// Mitsubishi GX Works2 project: BookEX6_23 Arithmetic   PLC: Q13UDV

// global labels: Global
VAR_GLOBAL
  bVar0 AT M5000 : BOOL;
  abArray0 AT M5010 : ARRAY [0..49] OF BOOL;
  sStr0 AT D5000 : STRING[199];
  sStr1 AT D5100 : STRING[199];
  sStr2 AT D5200 : STRING[199];
  sStr3 AT D5300 : STRING[199];
  sStr4 AT D5400 : STRING[199];
  sStr5 AT D5500 : STRING[199];
  sStr6 AT D5600 : STRING[199];
  sStr7 AT D5700 : STRING[199];
  sStr8 AT D5800 : STRING[199];
  sStr9 AT D5900 : STRING[199];
  iVar0 AT D4500 : INT;
  iVar1 AT D4501 : INT;
  iVar2 AT D4502 : INT;
  iVar3 AT D4503 : INT;
  iVar4 AT D4504 : INT;
  iVar5 AT D4505 : INT;
  iVar6 AT D4506 : INT;
  iVar7 AT D4507 : INT;
  iVar8 AT D4508 : INT;
  iVar9 AT D4509 : INT;
  dVar0 AT D4510 : DINT;
  dVar1 AT D4512 : DINT;
  dVar2 AT D4514 : DINT;
  dVar3 AT D4516 : DINT;
  dVar4 AT D4518 : DINT;
  dVar5 AT D4520 : DINT;
  dVar6 AT D4522 : DINT;
  dVar7 AT D4524 : DINT;
  dVar8 AT D4526 : DINT;
  dVar9 AT D4528 : DINT;
  wVar0 AT D4530 : WORD;
  wVar1 AT D4531 : WORD;
  wVar2 AT D4532 : WORD;
  wVar3 AT D4533 : WORD;
  wVar4 AT D4534 : WORD;
  wVar5 AT D4535 : WORD;
  wVar6 AT D4536 : WORD;
  wVar7 AT D4537 : WORD;
  wVar8 AT D4538 : WORD;
  wVar9 AT D4539 : WORD;
  dwVar0 AT D4540 : DWORD;
  dwVar1 AT D4542 : DWORD;
  dwVar2 AT D4544 : DWORD;
  dwVar3 AT D4546 : DWORD;
  dwVar4 AT D4548 : DWORD;
  dwVar5 AT D4550 : DWORD;
  dwVar6 AT D4552 : DWORD;
  dwVar7 AT D4554 : DWORD;
  dwVar8 AT D4556 : DWORD;
  dwVar9 AT D4558 : DWORD;
  fsVar0 AT D4560 : REAL;
  fsVar1 AT D4562 : REAL;
  fsVar2 AT D4564 : REAL;
  fsVar3 AT D4566 : REAL;
  fsVar4 AT D4568 : REAL;
  fsVar5 AT D4570 : REAL;
  fsVar6 AT D4572 : REAL;
  fsVar7 AT D4574 : REAL;
  fsVar8 AT D4576 : REAL;
  fsVar9 AT D4578 : REAL;
  fdVar0 AT D4580 : LREAL;
  tTime0 AT D4620 : TIME;
  tTime1 AT D4622 : TIME;
  tTime2 AT D4624 : TIME;
  tTime3 AT D4626 : TIME;
  tTime4 AT D4628 : TIME;
  tTime5 AT D4630 : TIME;
  tTime6 AT D4632 : TIME;
  tTime7 AT D4634 : TIME;
  tTime8 AT D4636 : TIME;
  tTime9 AT D4638 : TIME;
  tTime10 AT D4640 : TIME;
  bVar1 AT M5001 : BOOL;
  bVar2 AT M5002 : BOOL;
  bVar3 AT M5003 : BOOL;
  bVar4 AT M5004 : BOOL;
  bVar5 AT M5005 : BOOL;
  bVar6 AT M5006 : BOOL;
  bVar7 AT M5007 : BOOL;
  bVar8 AT M5008 : BOOL;
  bVar9 AT M5009 : BOOL;
  abArray1 AT M5060 : ARRAY [0..49] OF BOOL;
  abArray2 AT M5110 : ARRAY [0..49] OF BOOL;
  abArray3 AT M5160 : ARRAY [0..49] OF BOOL;
  abArray4 AT M5210 : ARRAY [0..49] OF BOOL;
  abArray5 AT M5260 : ARRAY [0..49] OF BOOL;
  abArray6 AT M5310 : ARRAY [0..49] OF BOOL;
  abArray7 AT M5360 : ARRAY [0..49] OF BOOL;
  abArray8 AT M5410 : ARRAY [0..49] OF BOOL;
  abArray9 AT M5460 : ARRAY [0..49] OF BOOL;
  fdVar1 AT D4584 : LREAL;
  fdVar2 AT D4588 : LREAL;
  fdVar3 AT D4592 : LREAL;
  fdVar4 AT D4596 : LREAL;
  fdVar5 AT D4600 : LREAL;
  fdVar6 AT D4604 : LREAL;
  fdVar7 AT D4608 : LREAL;
  fdVar8 AT D4612 : LREAL;
  fdVar9 AT D4616 : LREAL;
  afsPen0 AT D2000 : ARRAY [0..499] OF REAL;
  afsPen1 AT D3000 : ARRAY [0..499] OF REAL;
END_VAR
// user libraries (not included): HMI

PROGRAM ExAddSub2
VAR
  HMI20_1 : HMI20;
END_VAR
(* structured ladder/FBD written out as ST: instructions are called as NAME(EN, inputs, outputs); _pN, _eN, _tN stand for wires *)
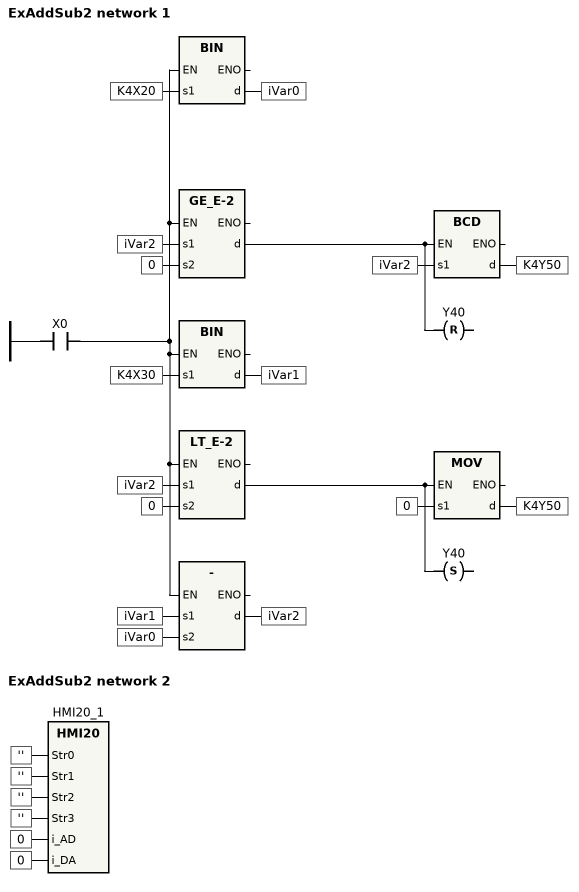
(* network 1 *)
BIN(X0, K4X20, iVar0);
BIN(X0, K4X30, iVar1);
-(X0, iVar1, iVar0, iVar2);
GE_E(X0, iVar2, 0, _t1);
BCD(_t1, iVar2, K4Y50);
RST(_t1, Y40);
LT_E(X0, iVar2, 0, _t2);
SET(_t2, Y40);
MOV(_t2, 0, K4Y50);
(* network 2 *)
HMI20_1(Str0 := '', Str1 := '', Str2 := '', Str3 := '', i_AD := 0, i_DA := 0);
END_PROGRAM

PROGRAM ExB
VAR
  wVar20 : WORD;
  wVar21 : WORD;
  wVar22 : WORD;
  wVar23 : WORD;
  wVar24 : WORD;
  wVar25 : WORD;
  wVar26 : WORD;
  wVar27 : WORD;
  wVar28 : WORD;
  wVar29 : WORD;
  dwVar20 : DWORD;
  dwVar21 : DWORD;
  dwVar22 : DWORD;
  dwVar23 : DWORD;
  dwVar24 : DWORD;
  dwVar25 : DWORD;
  dwVar26 : DWORD;
  dwVar27 : DWORD;
  dwVar28 : DWORD;
  dwVar29 : DWORD;
  awVar0 : ARRAY [0..1] OF WORD;
  awVar1 : ARRAY [0..1] OF WORD;
  awVar2 : ARRAY [0..3] OF WORD;
  awVar3 : ARRAY [0..3] OF WORD;
  adwVar3 : ARRAY [0..1] OF DWORD;
END_VAR
(* structured ladder/FBD written out as ST: instructions are called as NAME(EN, inputs, outputs); _pN, _eN, _tN stand for wires *)
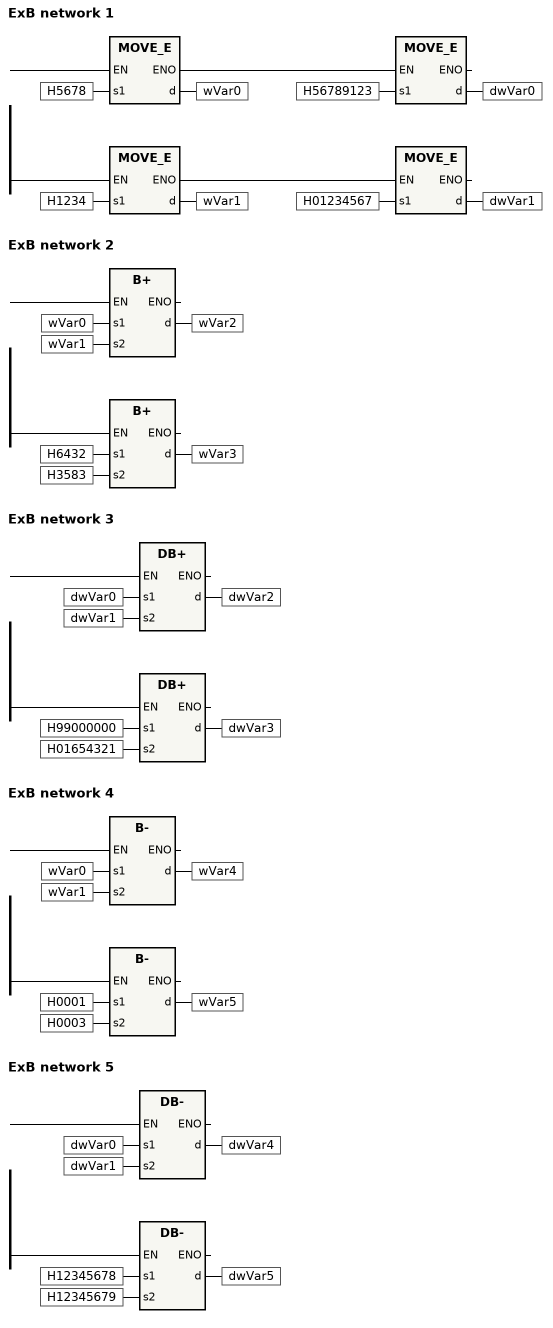
(* network 1 *)
_e1 := MOVE_E(TRUE, H5678, wVar0);
MOVE_E(_e1, H56789123, dwVar0);
_e2 := MOVE_E(TRUE, H1234, wVar1);
MOVE_E(_e2, H01234567, dwVar1);
(* network 2 *)
B+(TRUE, wVar0, wVar1, wVar2);
B+(TRUE, H6432, H3583, wVar3);
(* network 3 *)
DB+(TRUE, dwVar0, dwVar1, dwVar2);
DB+(TRUE, H99000000, H01654321, dwVar3);
(* network 4 *)
B-(TRUE, wVar0, wVar1, wVar4);
B-(TRUE, H0001, H0003, wVar5);
(* network 5 *)
DB-(TRUE, dwVar0, dwVar1, dwVar4);
DB-(TRUE, H12345678, H12345679, dwVar5);
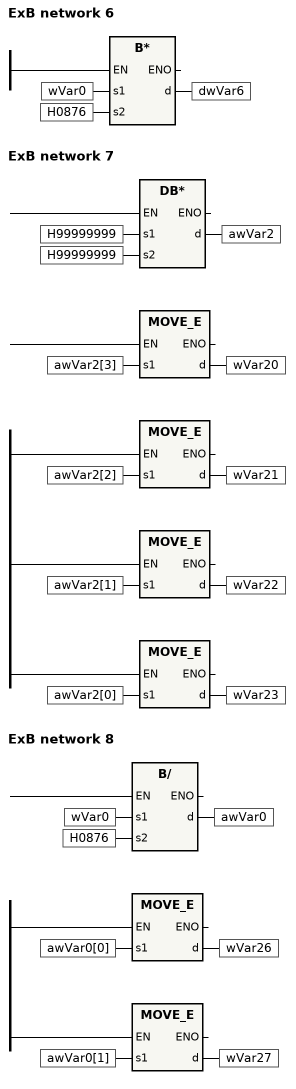
(* network 6 *)
B*(TRUE, wVar0, H0876, dwVar6);
(* network 7 *)
DB*(TRUE, H99999999, H99999999, awVar2);
MOVE_E(TRUE, awVar2[3], wVar20);
MOVE_E(TRUE, awVar2[2], wVar21);
MOVE_E(TRUE, awVar2[1], wVar22);
MOVE_E(TRUE, awVar2[0], wVar23);
(* network 8 *)
B/(TRUE, wVar0, H0876, awVar0);
MOVE_E(TRUE, awVar0[0], wVar26);
MOVE_E(TRUE, awVar0[1], wVar27);
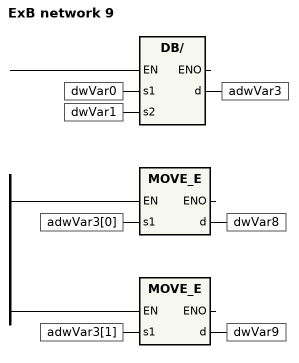
(* network 9 *)
DB/(TRUE, dwVar0, dwVar1, adwVar3);
MOVE_E(TRUE, adwVar3[0], dwVar8);
MOVE_E(TRUE, adwVar3[1], dwVar9);
END_PROGRAM

PROGRAM ExBK
VAR
  Mov4INT_1 : Mov4INT;
  Mov4INT_2 : Mov4INT;
END_VAR
(* structured ladder/FBD written out as ST: instructions are called as NAME(EN, inputs, outputs); _pN, _eN, _tN stand for wires *)
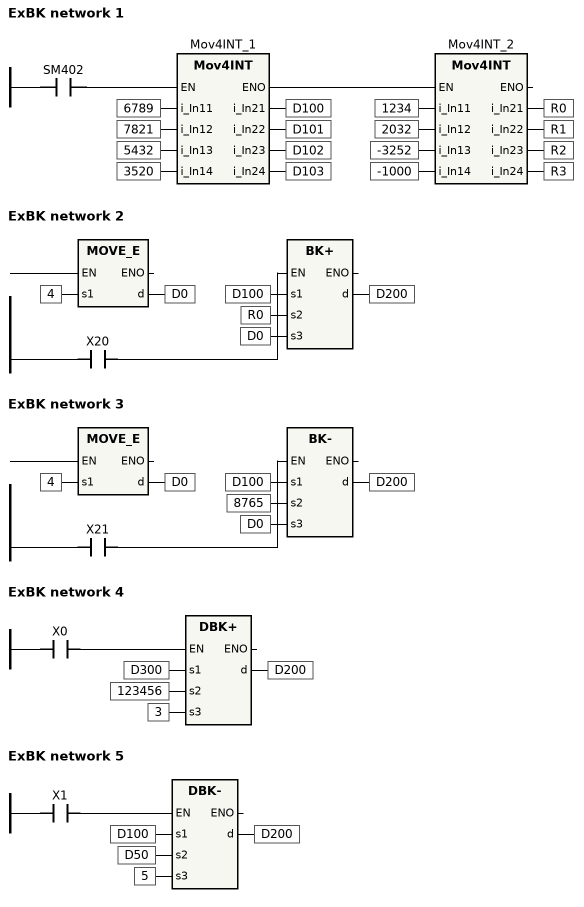
(* network 1 *)
Mov4INT_1(EN := SM402, i_In11 := 6789, i_In12 := 7821, i_In13 := 5432, i_In14 := 3520, i_In21 => D100, i_In22 => D101, i_In23 => D102, i_In24 => D103);
Mov4INT_2(EN := Mov4INT_1.ENO, i_In11 := 1234, i_In12 := 2032, i_In13 := -3252, i_In14 := -1000, i_In21 => R0, i_In22 => R1, i_In23 => R2, i_In24 => R3);
(* network 2 *)
MOVE_E(TRUE, 4, D0);
BK+(X20, D100, R0, D0, D200);
(* network 3 *)
MOVE_E(TRUE, 4, D0);
BK-(X21, D100, 8765, D0, D200);
(* network 4 *)
DBK+(X0, D300, 123456, 3, D200);
(* network 5 *)
DBK-(X1, D100, D50, 5, D200);
END_PROGRAM

PROGRAM ExIncDec
(* structured ladder/FBD written out as ST: instructions are called as NAME(EN, inputs, outputs); _pN, _eN, _tN stand for wires *)
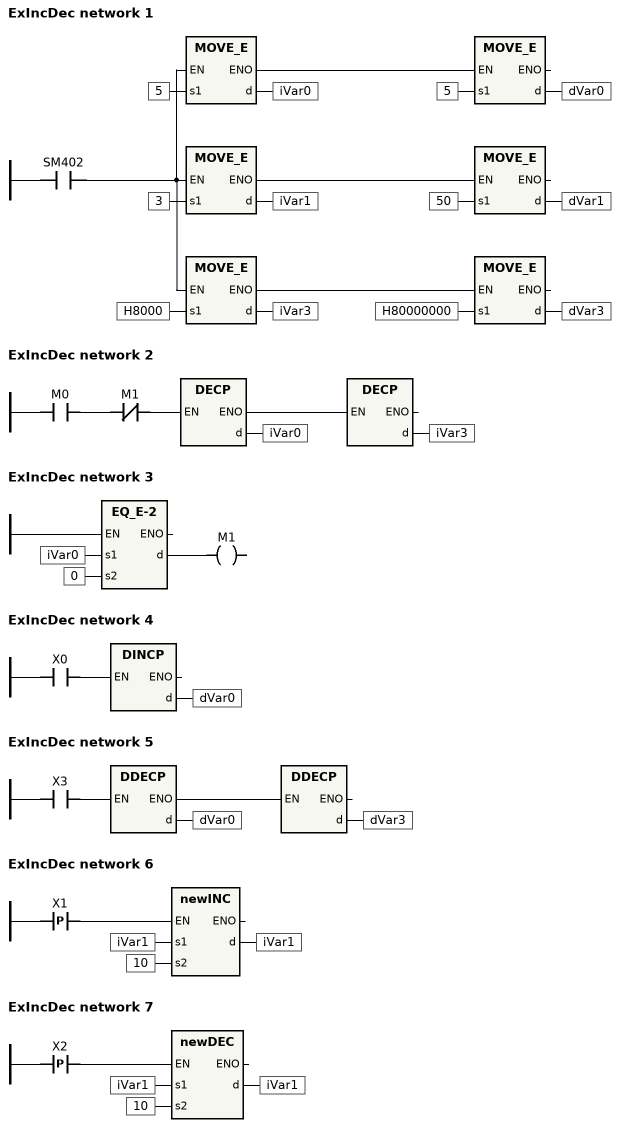
(* network 1 *)
_e1 := MOVE_E(SM402, 5, iVar0);
MOVE_E(_e1, 5, dVar0);
_e2 := MOVE_E(SM402, 3, iVar1);
MOVE_E(_e2, 50, dVar1);
_e3 := MOVE_E(SM402, H8000, iVar3);
MOVE_E(_e3, H80000000, dVar3);
(* network 2 *)
_e1 := DECP(M0 AND NOT M1, iVar0);
DECP(_e1, iVar3);
(* network 3 *)
EQ_E(TRUE, iVar0, 0, _t1);
M1 := _t1;
(* network 4 *)
DINCP(X0, dVar0);
(* network 5 *)
_e1 := DDECP(X3, dVar0);
DDECP(_e1, dVar3);
(* network 6 *)
newINC(LDP(TRUE, X1), iVar1, 10, iVar1);
(* network 7 *)
newDEC(LDP(TRUE, X2), iVar1, 10, iVar1);
END_PROGRAM

PROGRAM ExMulDiv
VAR
  iVar20 : INT;
  iVar21 : INT;
  iVar22 : INT;
  iVar23 : INT;
  iVar24 : INT;
  iVar25 : INT;
  iVar26 : INT;
  iVar27 : INT;
  iVar28 : INT;
  iVar29 : INT;
  dVar20 : DINT;
  dVar21 : DINT;
  dVar22 : DINT;
  dVar23 : DINT;
  dVar24 : DINT;
  dVar25 : DINT;
  dVar26 : DINT;
  dVar27 : DINT;
  dVar28 : DINT;
  dVar29 : DINT;
  aiVar0 : ARRAY [0..1] OF INT;
  aiVar1 : ARRAY [0..1] OF INT;
  aiVar2 : ARRAY [0..2] OF INT;
  awVar0 : ARRAY [0..1] OF WORD;
  awVar1 : ARRAY [0..1] OF WORD;
  awVar2 : ARRAY [0..3] OF WORD;
  awVar3 : ARRAY [0..3] OF WORD;
  adwVar3 : ARRAY [0..1] OF DWORD;
  adVar0 : ARRAY [0..1] OF DINT;
  adVar1 : ARRAY [0..1] OF DINT;
  adVar2 : ARRAY [0..1] OF DINT;
  adVar3 : ARRAY [0..1] OF DINT;
  adVar4 : ARRAY [0..1] OF DINT;
END_VAR
(* structured ladder/FBD written out as ST: instructions are called as NAME(EN, inputs, outputs); _pN, _eN, _tN stand for wires *)
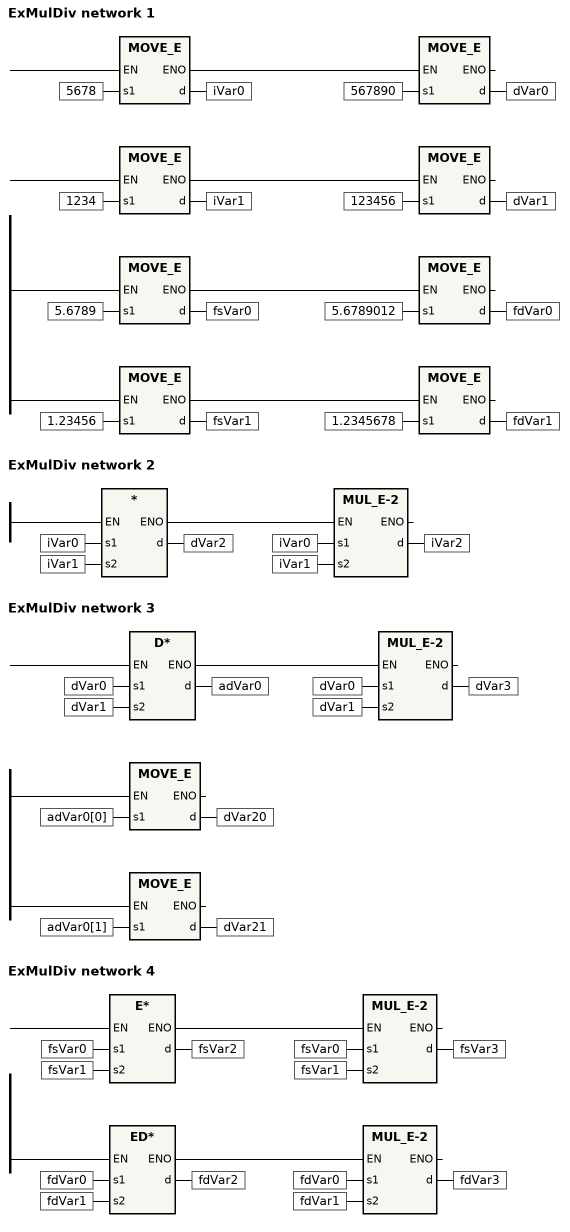
(* network 1 *)
_e1 := MOVE_E(TRUE, 5678, iVar0);
MOVE_E(_e1, 567890, dVar0);
_e2 := MOVE_E(TRUE, 1234, iVar1);
MOVE_E(_e2, 123456, dVar1);
_e3 := MOVE_E(TRUE, 5.6789, fsVar0);
MOVE_E(_e3, 5.6789012, fdVar0);
_e4 := MOVE_E(TRUE, 1.23456, fsVar1);
MOVE_E(_e4, 1.2345678, fdVar1);
(* network 2 *)
_e1 := *(TRUE, iVar0, iVar1, dVar2);
MUL_E(_e1, iVar0, iVar1, iVar2);
(* network 3 *)
_e1 := D*(TRUE, dVar0, dVar1, adVar0);
MUL_E(_e1, dVar0, dVar1, dVar3);
MOVE_E(TRUE, adVar0[0], dVar20);
MOVE_E(TRUE, adVar0[1], dVar21);
(* network 4 *)
_e1 := E*(TRUE, fsVar0, fsVar1, fsVar2);
MUL_E(_e1, fsVar0, fsVar1, fsVar3);
_e2 := ED*(TRUE, fdVar0, fdVar1, fdVar2);
MUL_E(_e2, fdVar0, fdVar1, fdVar3);
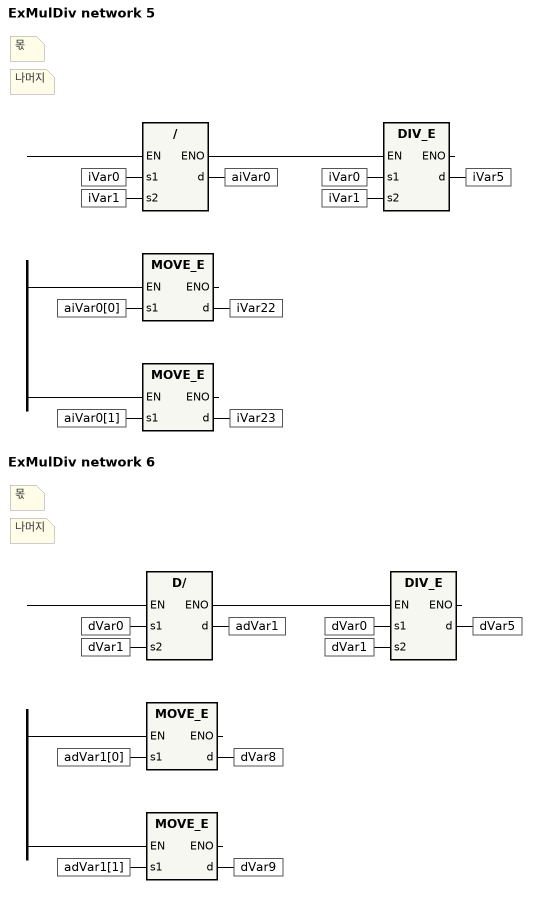
(* network 5 *)
(* 몫 *)
(* 나머지 *)
_e1 := /(TRUE, iVar0, iVar1, aiVar0);
DIV_E(_e1, iVar0, iVar1, iVar5);
MOVE_E(TRUE, aiVar0[0], iVar22);
MOVE_E(TRUE, aiVar0[1], iVar23);
(* network 6 *)
(* 몫 *)
(* 나머지 *)
_e1 := D/(TRUE, dVar0, dVar1, adVar1);
DIV_E(_e1, dVar0, dVar1, dVar5);
MOVE_E(TRUE, adVar1[0], dVar8);
MOVE_E(TRUE, adVar1[1], dVar9);
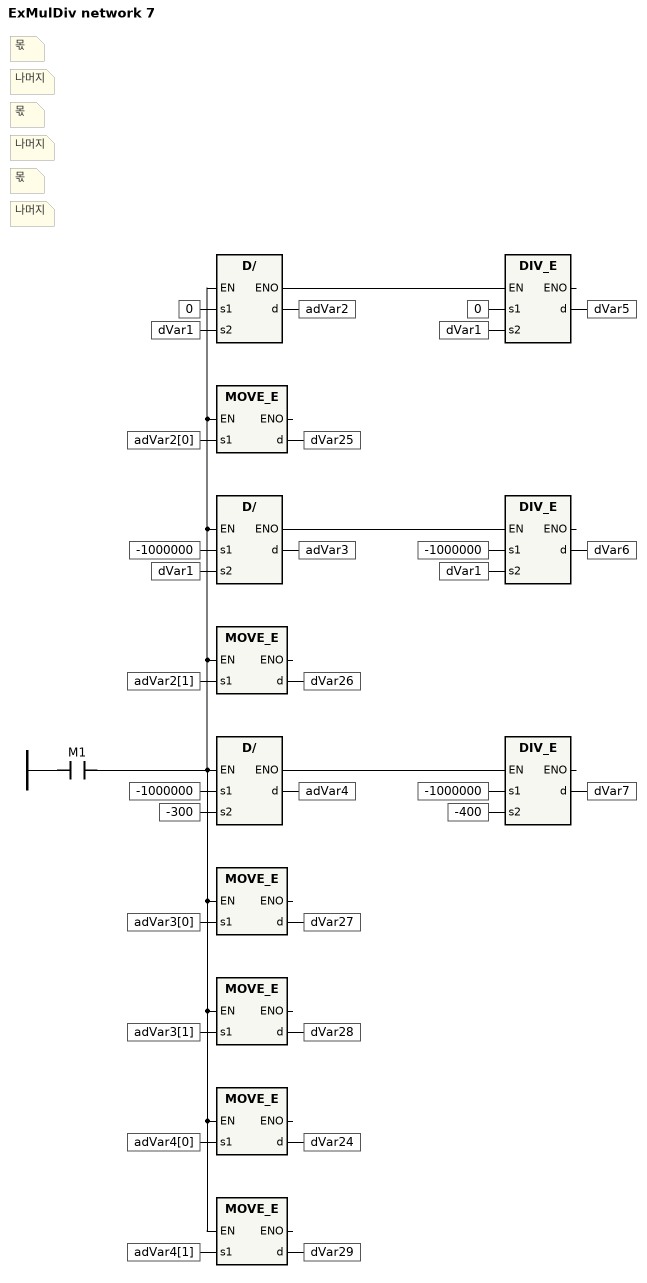
(* network 7 *)
(* 몫 *)
(* 나머지 *)
(* 몫 *)
(* 나머지 *)
(* 몫 *)
(* 나머지 *)
_e1 := D/(M1, 0, dVar1, adVar2);
DIV_E(_e1, 0, dVar1, dVar5);
MOVE_E(M1, adVar2[0], dVar25);
MOVE_E(M1, adVar2[1], dVar26);
_e2 := D/(M1, -1000000, dVar1, adVar3);
DIV_E(_e2, -1000000, dVar1, dVar6);
MOVE_E(M1, adVar3[0], dVar27);
MOVE_E(M1, adVar3[1], dVar28);
_e3 := D/(M1, -1000000, -300, adVar4);
DIV_E(_e3, -1000000, -400, dVar7);
MOVE_E(M1, adVar4[0], dVar24);
MOVE_E(M1, adVar4[1], dVar29);
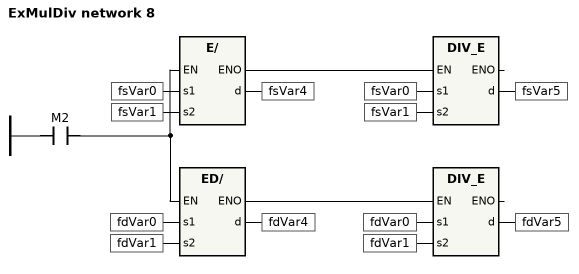
(* network 8 *)
_e1 := E/(M2, fsVar0, fsVar1, fsVar4);
DIV_E(_e1, fsVar0, fsVar1, fsVar5);
_e2 := ED/(M2, fdVar0, fdVar1, fdVar4);
DIV_E(_e2, fdVar0, fdVar1, fdVar5);
END_PROGRAM

PROGRAM ExString
(* structured ladder/FBD written out as ST: instructions are called as NAME(EN, inputs, outputs); _pN, _eN, _tN stand for wires *)
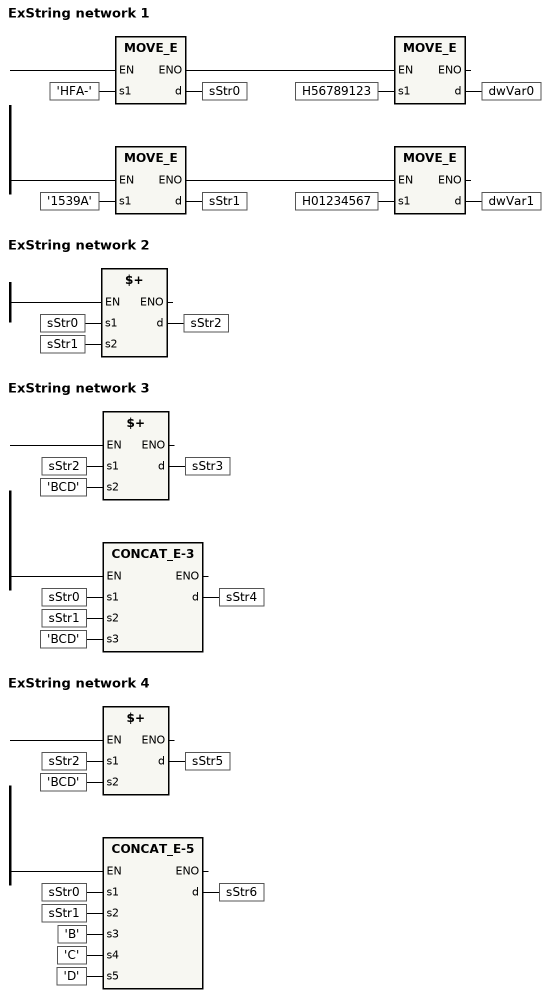
(* network 1 *)
_e1 := MOVE_E(TRUE, 'HFA-', sStr0);
MOVE_E(_e1, H56789123, dwVar0);
_e2 := MOVE_E(TRUE, '1539A', sStr1);
MOVE_E(_e2, H01234567, dwVar1);
(* network 2 *)
$+(TRUE, sStr0, sStr1, sStr2);
(* network 3 *)
$+(TRUE, sStr2, 'BCD', sStr3);
CONCAT_E(TRUE, sStr0, sStr1, 'BCD', sStr4);
(* network 4 *)
$+(TRUE, sStr2, 'BCD', sStr5);
CONCAT_E(TRUE, sStr0, sStr1, 'B', 'C', 'D', sStr6);
END_PROGRAM

FUNCTION newDEC
VAR_INPUT
  i_IN : INT;
  i_Max : INT;
END_VAR
VAR
  ix : INT;
END_VAR
;
ix := i_IN - 1;
IF ix < 0 THEN
	ix := i_Max;
END_IF;
newDEC := ix;
END_FUNCTION

FUNCTION newINC
VAR_INPUT
  i_IN : INT;
  i_Max : INT;
END_VAR
VAR
  ix : INT;
END_VAR
;
ix := i_IN + 1;
IF ix > i_Max THEN
	ix := 0;
END_IF;
newINC := ix;
END_FUNCTION

PROGRAM ExIncDec2
(* structured ladder/FBD written out as ST: instructions are called as NAME(EN, inputs, outputs); _pN, _eN, _tN stand for wires *)
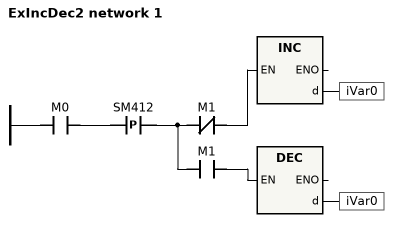
(* network 1 *)
_p1 := M0 AND LDP(TRUE, SM412);
INC(_p1 AND NOT M1, iVar0);
DEC(_p1 AND M1, iVar0);
END_PROGRAM

PROGRAM ExAddSub
VAR
  iVar20 : INT;
  iVar21 : INT;
  iVar22 : INT;
  iVar23 : INT;
  iVar24 : INT;
  iVar25 : INT;
  iVar26 : INT;
  iVar27 : INT;
  iVar28 : INT;
  iVar29 : INT;
  dVar20 : DINT;
  dVar21 : DINT;
  dVar22 : DINT;
  dVar23 : DINT;
  dVar24 : DINT;
  dVar25 : DINT;
  dVar26 : DINT;
  dVar27 : DINT;
  dVar28 : DINT;
  dVar29 : DINT;
  HMI05_1 : HMI05;
END_VAR
(* structured ladder/FBD written out as ST: instructions are called as NAME(EN, inputs, outputs); _pN, _eN, _tN stand for wires *)
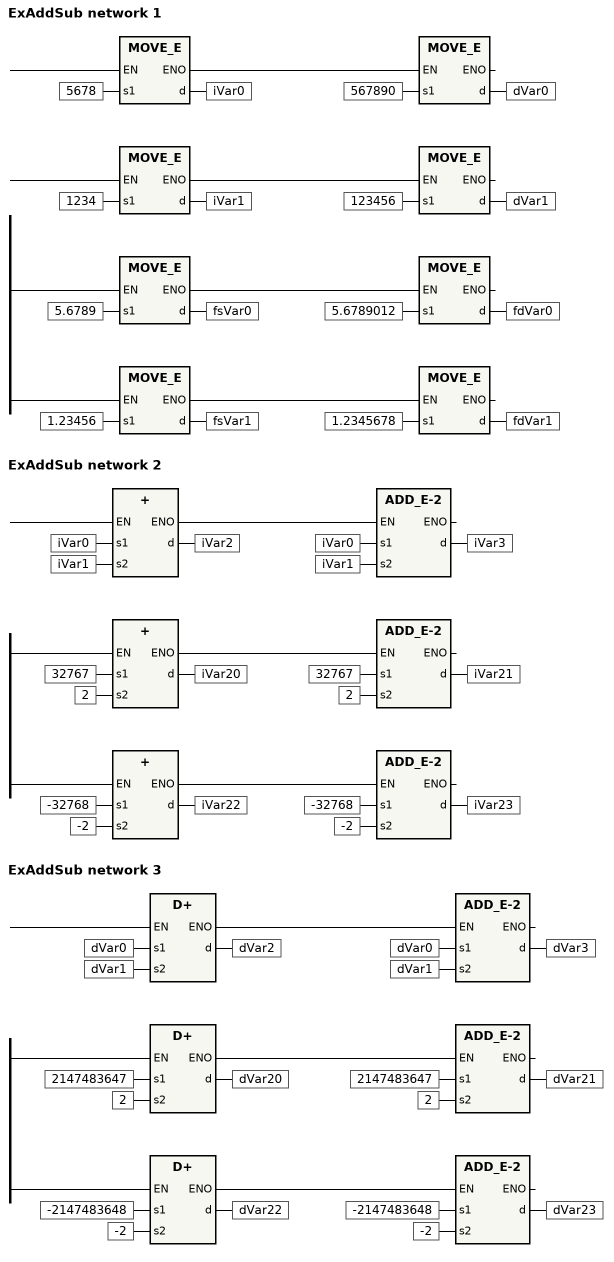
(* network 1 *)
_e1 := MOVE_E(TRUE, 5678, iVar0);
MOVE_E(_e1, 567890, dVar0);
_e2 := MOVE_E(TRUE, 1234, iVar1);
MOVE_E(_e2, 123456, dVar1);
_e3 := MOVE_E(TRUE, 5.6789, fsVar0);
MOVE_E(_e3, 5.6789012, fdVar0);
_e4 := MOVE_E(TRUE, 1.23456, fsVar1);
MOVE_E(_e4, 1.2345678, fdVar1);
(* network 2 *)
_e1 := +(TRUE, iVar0, iVar1, iVar2);
ADD_E(_e1, iVar0, iVar1, iVar3);
_e2 := +(TRUE, 32767, 2, iVar20);
ADD_E(_e2, 32767, 2, iVar21);
_e3 := +(TRUE, -32768, -2, iVar22);
ADD_E(_e3, -32768, -2, iVar23);
(* network 3 *)
_e1 := D+(TRUE, dVar0, dVar1, dVar2);
ADD_E(_e1, dVar0, dVar1, dVar3);
_e2 := D+(TRUE, 2147483647, 2, dVar20);
ADD_E(_e2, 2147483647, 2, dVar21);
_e3 := D+(TRUE, -2147483648, -2, dVar22);
ADD_E(_e3, -2147483648, -2, dVar23);
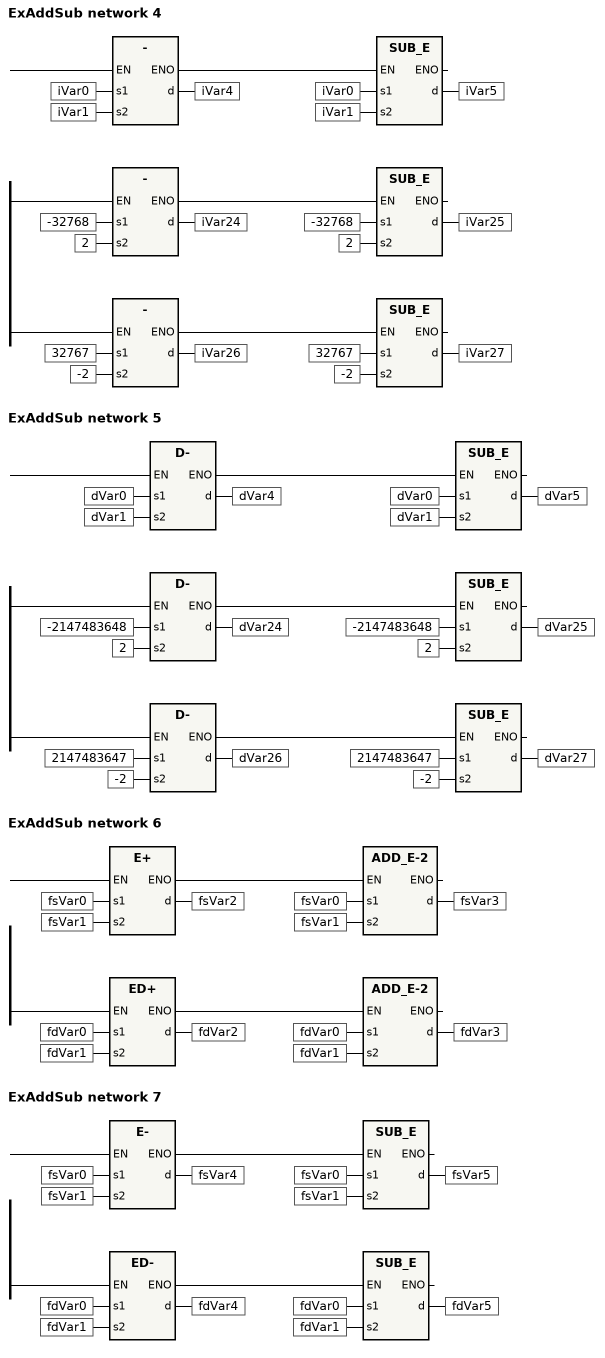
(* network 4 *)
_e1 := -(TRUE, iVar0, iVar1, iVar4);
SUB_E(_e1, iVar0, iVar1, iVar5);
_e2 := -(TRUE, -32768, 2, iVar24);
SUB_E(_e2, -32768, 2, iVar25);
_e3 := -(TRUE, 32767, -2, iVar26);
SUB_E(_e3, 32767, -2, iVar27);
(* network 5 *)
_e1 := D-(TRUE, dVar0, dVar1, dVar4);
SUB_E(_e1, dVar0, dVar1, dVar5);
_e2 := D-(TRUE, -2147483648, 2, dVar24);
SUB_E(_e2, -2147483648, 2, dVar25);
_e3 := D-(TRUE, 2147483647, -2, dVar26);
SUB_E(_e3, 2147483647, -2, dVar27);
(* network 6 *)
_e1 := E+(TRUE, fsVar0, fsVar1, fsVar2);
ADD_E(_e1, fsVar0, fsVar1, fsVar3);
_e2 := ED+(TRUE, fdVar0, fdVar1, fdVar2);
ADD_E(_e2, fdVar0, fdVar1, fdVar3);
(* network 7 *)
_e1 := E-(TRUE, fsVar0, fsVar1, fsVar4);
SUB_E(_e1, fsVar0, fsVar1, fsVar5);
_e2 := ED-(TRUE, fdVar0, fdVar1, fdVar4);
SUB_E(_e2, fdVar0, fdVar1, fdVar5);
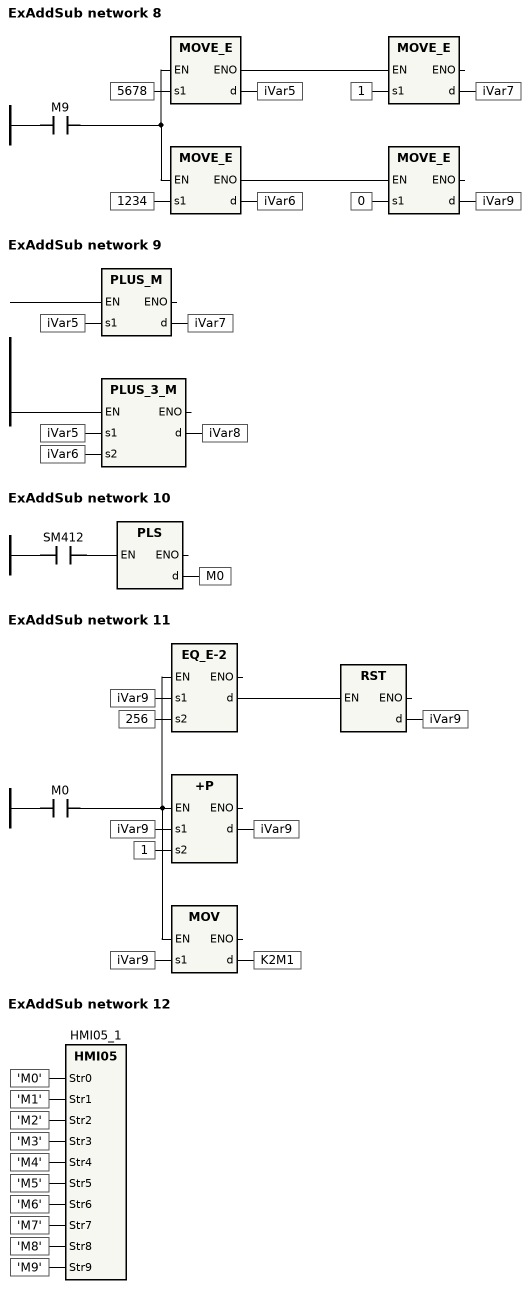
(* network 8 *)
_e1 := MOVE_E(M9, 5678, iVar5);
MOVE_E(_e1, 1, iVar7);
_e2 := MOVE_E(M9, 1234, iVar6);
MOVE_E(_e2, 0, iVar9);
(* network 9 *)
PLUS_M(TRUE, iVar5, iVar7);
PLUS_3_M(TRUE, iVar5, iVar6, iVar8);
(* network 10 *)
PLS(SM412, M0);
(* network 11 *)
+P(M0, iVar9, 1, iVar9);
MOV(M0, iVar9, K2M1);
EQ_E(M0, iVar9, 256, _t1);
RST(_t1, iVar9);
(* network 12 *)
HMI05_1(Str0 := 'M0', Str1 := 'M1', Str2 := 'M2', Str3 := 'M3', Str4 := 'M4', Str5 := 'M5', Str6 := 'M6', Str7 := 'M7', Str8 := 'M8', Str9 := 'M9');
END_PROGRAM
